// TIA Portal V19 export
FUNCTION_BLOCK "TYPIC_C501_IF_TRA"   // FB59, FBD
TITLE = TYPIC_C501_IF_TRA: Tracing
{ S7_Optimized_Access := 'TRUE' }
AUTHOR : OCOTECH
FAMILY : Typical
NAME : C501.705
// Logisch Object Besturing: C501.705
// stored: MemoryReserve 10, SetENOAutomatically false
   VAR_INPUT
      EXT_HW { ExternalAccessible := 'False'; ExternalVisible := 'False'; ExternalWritable := 'False'} : Bool;   // Sturings hardware (PLC) bewaking (1 = OK)
      IN_STO { ExternalAccessible := 'False'; ExternalVisible := 'False'; ExternalWritable := 'False'} : Bool;   // Storing Tracing (1 = OK)
   END_VAR
   VAR_OUTPUT
      VAR_IF_TRA { ExternalAccessible := 'False'; ExternalVisible := 'False'; ExternalWritable := 'False'} : "C501_VAR_IF_TRA_TYPIC";   // Struct met alle variabelen naar bovenliggende functies
   END_VAR
   VAR
      STO { ExternalWritable := 'False'} : Struct   // Storingen
         A001 : Bool;   // Storing vorstbeveiliging
      END_STRUCT;
      VAR { ExternalWritable := 'False'} : Struct   // Variabelen
         EXT_HW { ExternalAccessible := 'False'; ExternalVisible := 'False'} : Bool;   // Sturings hardware (PLC) in storing
      END_STRUCT;
   END_VAR
BEGIN

REGION Network 1: START
END_REGION

REGION Network 2: +++ Storingen +++
   // Verwerken van de storingsmeldingen (inputs).
END_REGION

REGION Network 3: Storing A001: Storing vorstbeveiliging
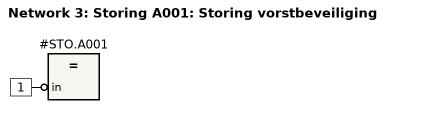
   #STO.A001 := NOT 1;
END_REGION

REGION Network 4 (SCL): EINDE
   // Variabelen van intern scada rakvlak naar outputs copieren
   #VAR_IF_TRA.EXT_HW := #VAR.EXT_HW;
   #VAR_IF_TRA.STO := #STO;
END_REGION
END_FUNCTION_BLOCK
